# EPICS IOC start-up script: examples/test/PSI/jinja2/loadPLCESS.iocsh
##############################################################################
## Need to install jinja2 and jinja2-cli:
## pip install -U Jinja2-cl
## pip install -U Jinja2
## pip install pyyaml

require ecmccfg,develop

##############################################################################
## Initiation:
epicsEnvSet("IOC" ,"$(IOC="IOC_TEST")")
epicsEnvSet("SCRIPTEXEC" ,"$(SCRIPTEXEC="iocshLoad")")

# run module startup.cmd (only needed at ESS  PSI auto call at require)
$(ECMCCFG_INIT="")$(SCRIPTEXEC) ${ecmccfg_DIR}startup.cmd, "IOC=$(IOC),ECMC_VER=6.3.2,MASTER_ID=-1"

#- ${SCRIPTEXEC} "${ECMC_CONFIG_ROOT}loadYamlPlc.cmd", "FILE=./plc1.ymal"
#- ${SCRIPTEXEC} "${ECMC_CONFIG_ROOT}loadYamlPlc.cmd" "FILE=./plc1.yaml
${SCRIPTEXEC} "${ECMC_CONFIG_ROOT}loadYamlPlc.cmd" "FILE=./plc1.yaml"

# go active
${SCRIPTEXEC} ${ECMC_CONFIG_ROOT}setAppMode.cmd
